% RSLogix 500 project project-one.rss, saved by version 8.30.00.16 %
PROJECT "UNTITLED"    % processor: Bul.1763 MicroLogix 1100 Series B %

PROGRAM FILES
  LAD 2 "MAIN"  4 rungs
  LAD 3 "D INPUT"  3 rungs
  LAD 4 "D OUTPUT"  3 rungs
  LAD 5 "CTRL LOGIC"  8 rungs

DATA FILES
  O0 OUTPUT  4 elements
  I1 INPUT  6 elements
  S2 STATUS  66 elements
  B3 BINARY  1 elements
  T4 TIMER  3 elements
  C5 COUNTER  1 elements
  R6 CONTROL  1 elements
  N7 INTEGER  1 elements
  F8 FLOAT  1 elements

LADDER 2 "MAIN"
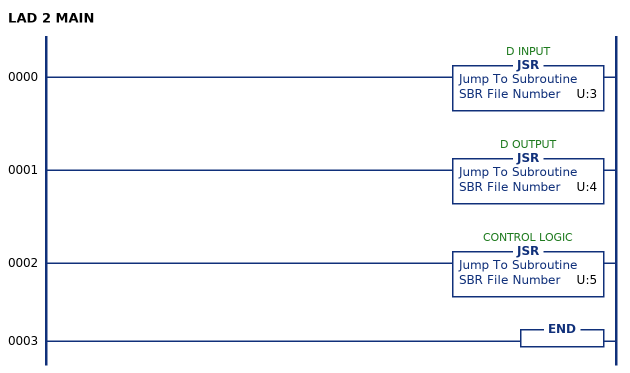
% Rung: 0 %
SOR JSR U:3 EOR
%   U:3  "D INPUT" %
% Rung: 1 %
SOR JSR U:4 EOR
%   U:4  "D OUTPUT" %
% Rung: 2 %
SOR JSR U:5 EOR
%   U:5  "CONTROL LOGIC" %
% Rung: 3 %
SOR END EOR

LADDER 3 "D INPUT"
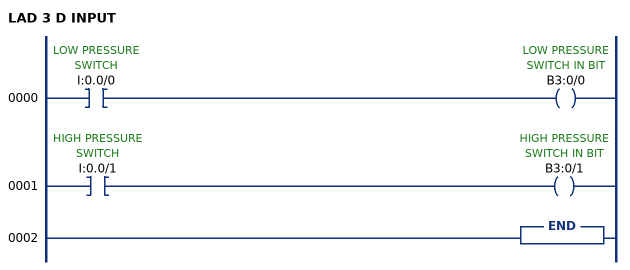
% Rung: 0 %
SOR XIC I:0.0/0 OTE B3:0/0 EOR
%   I:0.0/0  "LOW PRESSURE SWITCH" %
%   B3:0/0  "LOW PRESSURE SWITCH IN BIT" %
% Rung: 1 %
SOR XIC I:0.0/1 OTE B3:0/1 EOR
%   I:0.0/1  "HIGH PRESSURE SWITCH" %
%   B3:0/1  "HIGH PRESSURE SWITCH IN BIT" %
% Rung: 2 %
SOR END EOR

LADDER 4 "D OUTPUT"
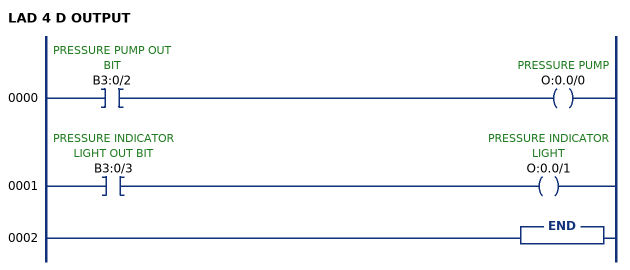
% Rung: 0 %
SOR XIC B3:0/2 OTE O:0.0/0 EOR
%   B3:0/2  "PRESSURE PUMP OUT BIT" %
%   O:0.0/0  "PRESSURE PUMP" %
% Rung: 1 %
SOR XIC B3:0/3 OTE O:0.0/1 EOR
%   B3:0/3  "PRESSURE INDICATOR LIGHT OUT BIT" %
%   O:0.0/1  "PRESSURE INDICATOR LIGHT" %
% Rung: 2 %
SOR END EOR

LADDER 5 "CTRL LOGIC"
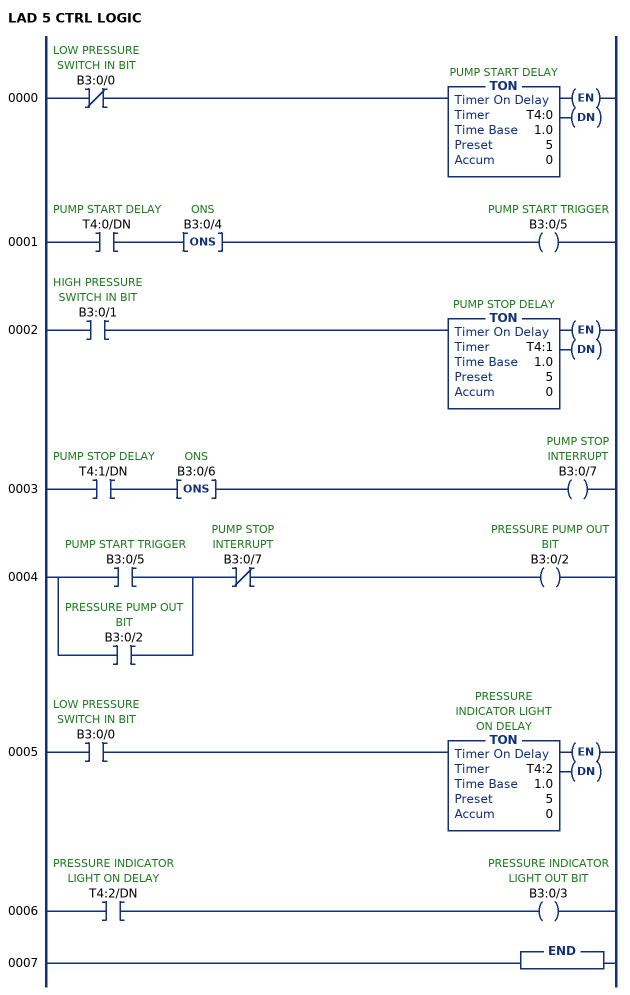
% Rung: 0 %
SOR XIO B3:0/0 TON T4:0 1.0 5 0 EOR
%   B3:0/0  "LOW PRESSURE SWITCH IN BIT" %
%   T4:0  "PUMP START DELAY" %
% Rung: 1 %
SOR XIC T4:0/DN ONS B3:0/4 OTE B3:0/5 EOR
%   T4:0  "PUMP START DELAY" %
%   B3:0/4  "ONS" %
%   B3:0/5  "PUMP START TRIGGER" %
% Rung: 2 %
SOR XIC B3:0/1 TON T4:1 1.0 5 0 EOR
%   B3:0/1  "HIGH PRESSURE SWITCH IN BIT" %
%   T4:1  "PUMP STOP DELAY" %
% Rung: 3 %
SOR XIC T4:1/DN ONS B3:0/6 OTE B3:0/7 EOR
%   T4:1  "PUMP STOP DELAY" %
%   B3:0/6  "ONS" %
%   B3:0/7  "PUMP STOP INTERRUPT" %
% Rung: 4 %
SOR BST XIC B3:0/5 NXB XIC B3:0/2 BND XIO B3:0/7 OTE B3:0/2 EOR
%   B3:0/5  "PUMP START TRIGGER" %
%   B3:0/2  "PRESSURE PUMP OUT BIT" %
%   B3:0/7  "PUMP STOP INTERRUPT" %
% Rung: 5 %
SOR XIC B3:0/0 TON T4:2 1.0 5 0 EOR
%   B3:0/0  "LOW PRESSURE SWITCH IN BIT" %
%   T4:2  "PRESSURE INDICATOR LIGHT ON DELAY" %
% Rung: 6 %
SOR XIC T4:2/DN OTE B3:0/3 EOR
%   T4:2  "PRESSURE INDICATOR LIGHT ON DELAY" %
%   B3:0/3  "PRESSURE INDICATOR LIGHT OUT BIT" %
% Rung: 7 %
SOR END EOR

DATA TABLE (non-zero values as saved)
DATA T4
% .PRE .ACC %
% T4:0 % 5 0
% T4:1 % 5 0
% T4:2 % 5 0
